FUNCTION_BLOCK RunInitClamperAndIndexer EXTENDS RunUnitGeneric
VAR_INPUT
	indexer : POINTER TO RunPnueIndexer;
	clampers : ARRAY[0..1] OF POINTER TO RunClamper;
	aoi : POINTER TO RunAoiInspectionV1;
	loader : POINTER TO runloading;
	
	okbin : POINTER TO RunBin;
	ngbin : POINTER TO RunBin;
END_VAR
VAR_OUTPUT
END_VAR
VAR
	nCounter : INT;
END_VAR

SUPER^();

CASE outputState OF 
	eSpecialStates.INITIAL_BEGIN:
		bSerialTransition:=TRUE;
		FOR nCounter:=0 TO 1 BY 1 DO
			bSerialTransition := bSerialTransition AND clampers[nCounter]^.Initialize();
		END_FOR
		bSerialTransition := bSerialTransition AND aoi^.Initialize();
		bSerialTransition := bSerialTransition AND loader^.Initialize();
		bSerialTransition := bSerialTransition AND okbin<>0 AND_THEN okbin^.Initialize();
		bSerialTransition := bSerialTransition AND ngbin<>0 AND_THEN ngbin^.Initialize();
	eSpecialStates.INITIAL_STATE_1:
		bSerialTransition := indexer^.Initialize();
		IF bSerialTransition THEN
			NextState := eSpecialStates.INITIAL_END;
		END_IF
	//-----------------------
	//	Working
	//-----------------------
	eSpecialStates.GENERIC_GROUP_START:
		FOR nCounter:=0 TO 1 BY 1 DO
			clampers[nCounter]^.NextState := eSpecialStates.GENERIC_GROUP_START;
		END_FOR
		aoi^.NextState := eSpecialStates.GENERIC_GROUP_START;
		indexer^.NextState := eSpecialStates.GENERIC_GROUP_START;
		loader^.NextState := eSpecialStates.GENERIC_GROUP_START;
		
		ngbin^.NextState := eSpecialStates.GENERIC_GROUP_START;
		okbin^.NextState := eSpecialStates.GENERIC_GROUP_START;
		
		bSerialTransition := TRUE; //into void state
END_CASE

END_FUNCTION_BLOCK

(* stored: Version 1.1.0.1, ProductVersion 3.1.4024.0
   POU RunInitClamperAndIndexer: Id {a648d874-3142-40b4-9333-4689f66f71a8}, SpecialFunc None *)
